FUNCTION F_DtToSqlTime : STRING
VAR_INPUT
	dtIn:TIMESTRUCT;
END_VAR
VAR
	s1:STRING;
END_VAR

s1:= WORD_TO_STRING(dtIn.wYear);
s1:=CONCAT(S1,'-');
S1:=CONCAT(S1,WORD_TO_STRING(dtIn.wMonth));
s1:=CONCAT(s1,'-');
s1:=CONCAT(S1,WORD_TO_STRING(dtIn.wDay));
s1:=CONCAT(s1,' ');
s1:=CONCAT(s1,WORD_TO_STRING(dtIN.wHour));
s1:=CONCAT(S1,':');
S1:=CONCAT(s1,WORD_TO_STRING(dtIN.wMinute));
s1:=CONCAT(s1,':');
s1:=CONCAT(s1,WORD_TO_STRING(dtIN.wSecond));

F_DtToSqlTime:=S1;

END_FUNCTION

(* stored: Version 1.1.0.1, ProductVersion 3.1.4024.12
   POU F_DtToSqlTime: Id {c84f2a71-a526-4dd1-a185-32578f9fc50d}, SpecialFunc None *)
